{attribute 'linkalways'} 
{attribute 'no_explicit_call' := 'This FB is a CLASS and must be accessed using methods or properties'}
{attribute 'enable_dynamic_creation'}
FUNCTION_BLOCK _ETcVnHoughMethod EXTENDS EnumDatatypeBase
VAR
	localData : ETcVnHoughMethod;
	activeData : REFERENCE TO ETcVnHoughMethod;
	enumBaseDatatype : _DINT(localData);
END_VAR

METHOD PRIVATE AddLocalEnumeration
VAR_INPUT
	Enumeration : T_MAXSTRING;
	Value : ETcVnHoughMethod;
END_VAR
AddEnumeration(Enumeration, Value);
END_METHOD

PROPERTY PUBLIC Address : PVOID
GET
Address := ADR(activeData);
END_GET
END_PROPERTY

METHOD PUBLIC ClearReference
VAR_INPUT
END_VAR
activeData REF= localData;
SetBaseDatatypeReference();
END_METHOD

METHOD PUBLIC Clone : I_Datatype
VAR
    pClone : POINTER TO _ETcVnHoughMethod;
END_VAR
pClone := __NEW(_ETcVnHoughMethod(InitialValue := Value));
Clone := pClone^;
END_METHOD

METHOD FB_init : BOOL
VAR_INPUT
	bInitRetains : BOOL; // if TRUE, the retain variables are initialized (warm start / cold start)
	bInCopyCode : BOOL;  // if TRUE, the instance afterwards gets moved into the copy code (online change)
	InitialValue : ETcVnHoughMethod;
END_VAR
localData := InitialValue;
AddBaseDatatype(enumBaseDatatype);
ClearReference();

AddLocalEnumeration('TCVN_HM_STANDARD', ETcVnHoughMethod.TCVN_HM_STANDARD);
AddLocalEnumeration('TCVN_HM_PROBABILISTIC', ETcVnHoughMethod.TCVN_HM_PROBABILISTIC);
AddLocalEnumeration('TCVN_HM_MULTI_SCALE', ETcVnHoughMethod.TCVN_HM_MULTI_SCALE);
AddLocalEnumeration('TCVN_HM_GRADIENT', ETcVnHoughMethod.TCVN_HM_GRADIENT);
AddLocalEnumeration('TCVN_HM_GRADIENT_ALT', ETcVnHoughMethod.TCVN_HM_GRADIENT_ALT);
END_METHOD

PROPERTY PUBLIC Identifier : T_MAXSTRING
GET
Identifier := 'ETcVnHoughMethod';
END_GET
END_PROPERTY

METHOD IsEnumeratorValueEqual : BOOL
VAR_INPUT
	Enumerator : I_KeyValueForwardEnumerator;
END_VAR
VAR
	storedValue : ETcVnHoughMethod;
END_VAR
IF NOT Enumerator.TryGet(storedValue) THEN
	RETURN;
END_IF

IsEnumeratorValueEqual := storedValue = activeData;
END_METHOD

METHOD PUBLIC MakeReferenceTo
VAR_INPUT
	ReferenceTarget : REFERENCE TO ETcVnHoughMethod;
END_VAR
activeData REF= ReferenceTarget;
SetBaseDatatypeReference();
END_METHOD

METHOD PROTECTED SetBaseDatatypeReference
VAR_INPUT
END_VAR
enumBaseDatatype.MakeReferenceTo(activeData);
END_METHOD

PROPERTY PUBLIC Size : UDINT
GET
Size := SIZEOF(activeData);
END_GET
END_PROPERTY

METHOD TryMakeReferenceTo : BOOL
VAR_INPUT
	Target : I_Datatype;
END_VAR
VAR
	targetAsEnum : I_EnumDatatype;
	pTargetData : POINTER TO ETcVnHoughMethod;
END_VAR
IF NOT Target.TryResolveAsEnumDatatype(targetAsEnum) THEN
	RETURN;
END_IF

IF targetAsEnum.Identifier <> Identifier THEN
	RETURN;
END_IF

pTargetData := Target.Address;
activeData REF= pTargetData^;
SetBaseDatatypeReference();
TryMakeReferenceTo := TRUE;
END_METHOD

PROPERTY PUBLIC Value : ETcVnHoughMethod
GET
Value := activeData;
END_GET
SET
activeData := Value;
END_SET
END_PROPERTY

END_FUNCTION_BLOCK

(* stored: Version 1.1.0.1, ProductVersion 3.1.4024.12
   POU _ETcVnHoughMethod: Id {8e8e81ba-7bc2-0eb0-0aa6-b932849bfacf}, SpecialFunc None
   Folder Constructor: Id {825a3143-73ff-0ac0-1490-f66c3f30edf0}
   Folder Private: Id {2d7bfa7f-af78-0d27-2806-91775ddc4d78}
   Folder Protected: Id {9b798fd3-90ae-05b0-365e-a1b98ad5af53}
   Method AddLocalEnumeration: Id {d594f1db-523a-018c-35d2-fa9c98b06a13}
   Property Address: Id {3bf72501-bca5-08db-1472-f02db18d984c}
   Get Get: Id {c469a997-4aa4-0b77-35cb-7e927fcfdc53}
   Method ClearReference: Id {cc77b2af-f324-0c11-0e11-9c0044b817eb}
   Method Clone: Id {99b9c5a2-4592-00ba-38be-70f77148bf5b}
   Method FB_init: Id {85b8c148-50be-0f3c-04f1-9ec00b42c47f}
   Property Identifier: Id {ef6a9525-e29a-0146-3570-b249750796a0}
   Get Get: Id {4995b785-da1d-0562-2a96-340aa0c394cf}
   Method IsEnumeratorValueEqual: Id {0ff8d33d-0455-07cd-2d8b-48bbe6103a14}
   Method MakeReferenceTo: Id {61e4f5fd-7d7a-0ac8-0856-88fe62fb6b54}
   Method SetBaseDatatypeReference: Id {4466f6d5-3869-06cd-13c6-46cb809eb4c2}
   Property Size: Id {aa7d1303-17ee-08da-3e5e-b6ccde068d20}
   Get Get: Id {7e9e6cab-8613-0c04-06de-d9202120d4a8}
   Method TryMakeReferenceTo: Id {08816ede-525c-04d5-01e3-a256f8c9ca83}
   Property Value: Id {4d0326cc-7d48-044c-2c2a-505c12523b9f}
   Get Get: Id {376be4ff-3d15-09b4-3279-0d0e093ce550}
   Set Set: Id {f0803f8a-a67e-0d4c-0817-2ced4c3c41d7} *)
